FUNCTION_BLOCK FB_Level EXTENDS FB_Element
VAR_INPUT
	fbList:				FB_ListElement;
END_VAR
VAR_OUTPUT
END_VAR
VAR
END_VAR

SUPER^();

METHOD PROTECTED M_Aborting : BOOL (* Return*)
VAR
	nIndex: 	UINT;
END_VAR
M_Aborting:= TRUE;
WHILE nIndex < fbList.nLength DO
    IF fbList.M_Index(nIndex).M_Request(E_Request.Abort) THEN
		;
	ELSE
		M_Aborting:= FALSE;
	END_IF
	nIndex := nIndex + 1;
END_WHILE
END_METHOD

METHOD PUBLIC M_Attach : BOOL
VAR_INPUT
	iComponent:		I_Element;
END_VAR
fbList.M_Add(iComponent);
iComponent.P_Event.P_Logger:= fbEvent.P_Logger;
iComponent.P_Event.P_Observer.M_Attach(THIS^);
fbEvent.fbObserver.M_Attach(iComponent);
M_Attach:= TRUE;
END_METHOD

METHOD PUBLIC M_Detach : BOOL
VAR_INPUT
END_VAR
END_METHOD

METHOD PROTECTED M_Resetting : BOOL (* Return*)
VAR
	nIndex: 	UINT;
END_VAR
M_Resetting:= TRUE;
WHILE nIndex < fbList.nLength DO
    IF fbList.M_Index(nIndex).M_Request(E_Request.Reset) THEN
		;
	ELSE
		M_Resetting:= FALSE;
	END_IF
	nIndex := nIndex + 1;
END_WHILE
END_METHOD

METHOD PROTECTED M_Starting : BOOL (* Return*)
VAR
	nIndex: 	UINT;
END_VAR
M_Starting:= TRUE;
WHILE nIndex < fbList.nLength DO
    IF fbList.M_Index(nIndex).M_Request(E_Request.Start) THEN
		;
	ELSE
		M_Starting:= FALSE;
	END_IF
	nIndex := nIndex + 1;
END_WHILE
END_METHOD

METHOD PROTECTED M_Stopping : BOOL (* Return state complete*)
VAR
	nIndex: 	UINT;
END_VAR
M_Stopping:= TRUE;
WHILE nIndex < fbList.nLength DO
    IF fbList.M_Index(nIndex).M_Request(E_Request.Reset) THEN
		;
	ELSE
		M_Stopping:= FALSE;
	END_IF
	nIndex := nIndex + 1;
END_WHILE
END_METHOD

PROPERTY PUBLIC P_List : I_ListElement
GET
P_List:= fbList;
END_GET
END_PROPERTY

END_FUNCTION_BLOCK

(* stored: Version 1.1.0.1
   POU FB_Level: Id {cd8da5ab-5393-0aad-280e-8aa1aa48dea2}, SpecialFunc None
   Method M_Aborting: Id {104d8837-6bb5-0521-1173-730037e337c3}
   Method M_Attach: Id {0c962b9d-42f1-04de-310f-7afbe89f613e}
   Method M_Detach: Id {7aeefa55-b634-02b3-27c8-71b7445f7fa7}
   Method M_Resetting: Id {ae571459-9edd-0301-20e5-a7a9f4f76ff7}
   Method M_Starting: Id {7ad18ebf-7549-0791-216c-829f6009eac2}
   Method M_Stopping: Id {3af3bc97-6689-0cd0-087b-ea87e272f27c}
   Property P_List: Id {54577eeb-5f19-02a6-0647-7059c4555532}
   Get Get: Id {e32edb93-fe26-01ab-0e1d-a118b7b75f71} *)
